FUNCTION_BLOCK FB_Observer IMPLEMENTS InterfaceObserver
VAR_INPUT
END_VAR
VAR_OUTPUT
	job_event_report : JobEventReport;
END_VAR
VAR
END_VAR

METHOD subscribe_job_directory : BOOL
VAR_INPUT
	(* Represent reference to subscribed job object*)
	executor	: REFERENCE TO jobmgmt.FB_Executor;
END_VAR
VAR
	job_log : STRING;
END_VAR
job_log := CONCAT(job_log, 'JOB STRUCTURE');
IF executor.future <> 0 THEN
	job_log := CONCAT(job_log, '/ FUTURE_NAME :');
	job_log := CONCAT(job_log, executor.future.future_name);
	job_log := CONCAT(job_log, ',');
END_IF

job_log := CONCAT(job_log, 'JOB_ID');
job_log := CONCAT(job_log, ' : ');
job_log := CONCAT(job_log, executor.uid);

ADSLOGSTR(msgCtrlMask := ADSLOG_MSGTYPE_LOG, msgFmtStr := job_log, strArg := '');
END_METHOD

METHOD subscribe_job_event : BOOL
VAR_INPUT
	(* Subject of event*)
	subject	: T_MaxString;
	(* Job state before transition.*)
	old_state	: jobmgmt.E_FutureExecutionState;
	(* Job state after transition.*)
	new_state	: jobmgmt.E_FutureExecutionState;
	(* File-time at the time of transition.*)
	record_time	: jobmgmt.T_FILETIME64;
	(* Reference to job instance of which transition occurs.*)
	executor	: REFERENCE TO jobmgmt.FB_Executor;
END_VAR
VAR_INST
	fb_timezone_info : FB_GetTimeZoneInformation := (bExecute := TRUE);
END_VAR
VAR
	last_state : STRING;
	current_state : STRING;
	text : T_MaxString;
	container : InterfaceContainer;
	num_of_jobs : UINT;
END_VAR
last_state := TO_STRING(old_state);
current_state := TO_STRING(new_state);

IF __QUERYINTERFACE(executor.future, container) THEN
	num_of_jobs := container.num_of_jobs;
ELSE
	num_of_jobs := 0;
END_IF


IF __ISVALIDREF(executor) THEN
	fb_timezone_info();
	text := FILETIME64_TO_ISO8601(fileTime := record_time, nBias := DINT_TO_INT(fb_timezone_info.tzInfo.bias), bUTC := TRUE,nPrecision := 6);
	text := CONCAT(text, '	');
	text := CONCAT(text, subject);
	text := CONCAT(text, '	');
	text := CONCAT(text, TO_STRING(current_state));
	text := CONCAT(text, '	Err:');
	text := CONCAT(text, TO_STRING(executor.nErrorID));
	text := CONCAT(text, '		SubJob:');
	text := CONCAT(text, TO_STRING(num_of_jobs));
	text := CONCAT(text, '		Name:');
	text := CONCAT(text, executor.future.future_name);
	text := CONCAT(text, '		JobID:');
	text := CONCAT(text, executor.uid);
		
	ADSLOGSTR(msgCtrlMask := ADSLOG_MSGTYPE_LOG,
 			 msgFmtStr := text, 
			strArg := '');	
END_IF


job_event_report.future_name := executor.future.future_name;
job_event_report.job_id := executor.uid;
job_event_report.new_state := TO_STRING(new_state);
job_event_report.old_state := TO_STRING(old_state);
job_event_report.record_time := record_time;
job_event_report.subject := subject;

subscribe_job_event := TRUE;
END_METHOD

END_FUNCTION_BLOCK

(* stored: Version 1.1.0.1, ProductVersion 3.1.4024.12
   POU FB_Observer: Id {adc11630-587f-43db-9eda-5da3af2be89b}, SpecialFunc None
   Method subscribe_job_directory: Id {9fadc14a-702e-4d4c-9c8d-d3d1919e5052}
   Method subscribe_job_event: Id {4ef31f8a-7d23-4675-adf8-d567da162687} *)
